Fanuc KAREL source: CA0113.KL

-- PROVISIONAL review KL for V940-1; original PC SHA256 f2846a05208e82293c29ea2b9839217a6d33d7e8cb96e12588648d0b48dd8da7
-- Incomplete behavior may be omitted. Consult companion uncertainty JSON. Do not deploy.
PROGRAM CA0113
%NOLOCKGROUP
BEGIN
  -- V9_ZERO_TABLE_METADATA_HINT layout=0001; no indexed target words; source/name/runtime held
  -- UNRESOLVED_PC offsets 0-1; opcodes 7B
  -- UNRESOLVED_PC offsets 6-16; opcodes 2D,7F
  -- UNRESOLVED_PC offsets 21-25; opcodes 7F
  -- UNRESOLVED_PC offsets 30-37; opcodes 9C,23
  -- UNRESOLVED_PC offsets 42-49; opcodes 9D,23
  -- UNRESOLVED_PC offsets 54-65; opcodes 2E,23
  -- UNRESOLVED_PC offsets 70-77; opcodes 9D,23
  -- UNRESOLVED_PC offsets 82-91; opcodes 3F,75
  -- UNRESOLVED_PC offsets 96-110; opcodes 2E,22,9D,33,35
  -- UNRESOLVED_PC offsets 115-129; opcodes 2E,22,9D,33,35
  -- UNRESOLVED_PC offsets 134-149; opcodes 2E,22,32,35
  -- UNRESOLVED_PC offsets 154-169; opcodes 2E,22,32,35
  -- UNRESOLVED_PC offsets 174-208; opcodes 27,22,22,22,22,AA,23
  -- UNRESOLVED_PC offsets 213-217; opcodes 7F
END CA0113
